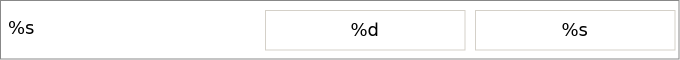
VISUALIZATION SingleRecipesParameterTypeInteger  // 680x60
VAR_IN_OUT
	stRecipeParameter : ST_VisuCtrlRecipeParameter;
END_VAR
    Textfield (265,10 200x40), "%d", text variable: stRecipeParameter.iValue
        OnMouseClick: write the text variable via VisuDialogs.Numpad
    Textfield (475,10 200x40), "%s", text variable: stRecipeParameter.sFileValue
    Textfield (5,8 250x40), "%s", text variable: stRecipeParameter.sName
END_VISUALIZATION

(* stored: Version 1.1.0.1, ProductVersion 3.1.4024.12
   Visu SingleRecipesParameterTypeInteger: Id {2484aab2-3358-4ab3-bbff-e2df100d33e1} *)
